(* IEC 61131-3 sources: IRIS-Project/LASAL CONTROL SOFTWARE/LasalProject_2025_09_25/Class/Automatic_Step_Settings, 1 file *)

(* ---- Automatic_Step_Settings.st ---- *)
(*!
<Class
	Name               = "Automatic_Step_Settings"
	Revision           = "0.0"
	RealtimeTask       = "false"
	CyclicTask         = "true"
	DefCyclictime      = "500 ms"
	BackgroundTask     = "false"
	Sigmatek           = "false"
	OSInterface        = "false"
	HighPriority       = "false"
	Automatic          = "false"
	UpdateMode         = "Prescan"
	SharedCommandTable = "true"
	Objectsize         = "(900,1020)">
	<Channels>
		<Server Name="ClassSvr" Visualized="false" Initialize="false" WriteProtected="true" Retentive="false"/>
		<Server Name="M1_Correction_Step" Visualized="false" Initialize="false" WriteProtected="false" Retentive="false"/>
		<Server Name="M3_Correction_Step" Visualized="false" Initialize="false" WriteProtected="false" Retentive="false"/>
		<Server Name="M4_Correction_Step" Visualized="false" Initialize="false" WriteProtected="false" Retentive="false"/>
		<Server Name="M5_ChargingCorrection_step_1" Visualized="false" Initialize="false" WriteProtected="false" Retentive="false"/>
		<Server Name="M5_ChargingCorrection_step_2" Visualized="false" Initialize="false" WriteProtected="false" Retentive="false"/>
		<Server Name="M5_ChargingCorrection_step_3" Visualized="false" Initialize="false" WriteProtected="false" Retentive="false"/>
		<Server Name="M5_DischargingCorrection_step" Visualized="false" Initialize="false" WriteProtected="false" Retentive="false"/>
		<Server Name="M5_IrradiationCorrection_step_1" Visualized="false" Initialize="false" WriteProtected="false" Retentive="false"/>
		<Server Name="M5_IrradiationCorrection_step_2" Visualized="false" Initialize="false" WriteProtected="false" Retentive="false"/>
		<Server Name="M5_IrradiationCorrection_step_3" Visualized="false" Initialize="false" WriteProtected="false" Retentive="false"/>
		<Client Name="c_M1_Correction_Step" Required="false" Internal="false"/>
		<Client Name="c_M3_Correction_Step" Required="true" Internal="false"/>
		<Client Name="c_M4_Correction_Step" Required="true" Internal="false"/>
		<Client Name="c_M5_ChargingCorrection_Step_1" Required="true" Internal="false"/>
		<Client Name="c_M5_ChargingCorrection_Step_2" Required="true" Internal="false"/>
		<Client Name="c_M5_ChargingCorrection_Step_3" Required="true" Internal="false"/>
		<Client Name="c_M5_DischargingCorrection_step" Required="true" Internal="false"/>
		<Client Name="c_M5_IrradiationCorrection_Step_1" Required="true" Internal="false"/>
		<Client Name="c_M5_IrradiationCorrection_Step_2" Required="true" Internal="false"/>
		<Client Name="c_M5_IrradiationCorrection_step_3" Required="true" Internal="false"/>
	</Channels>
	<Separators>
		<Servers>
			<SepChn Position="3"/>
			<SepChn Position="7"/>
			<SepChn Position="11"/>
			<SepChn Position="15"/>
			<SepChn Position="1"/>
			<SepChn Position="5"/>
		</Servers>
		<Clients>
			<SepChn Position="1"/>
			<SepChn Position="5"/>
			<SepChn Position="9"/>
			<SepChn Position="13"/>
			<SepChn Position="3"/>
		</Clients>
	</Separators>
</Class>
*)
Automatic_Step_Settings : CLASS
  //Servers:
	ClassSvr 	: SvrChCmd_DINT;
	M1_Correction_Step 	: SvrCh_DINT;
	M3_Correction_Step 	: SvrCh_DINT;
	M4_Correction_Step 	: SvrCh_DINT;
	M5_ChargingCorrection_step_1 	: SvrCh_DINT;
	M5_ChargingCorrection_step_2 	: SvrCh_DINT;
	M5_ChargingCorrection_step_3 	: SvrCh_DINT;
	M5_IrradiationCorrection_step_1 	: SvrCh_DINT;
	M5_IrradiationCorrection_step_2 	: SvrCh_DINT;
	M5_IrradiationCorrection_step_3 	: SvrCh_DINT;
	M5_DischargingCorrection_step 	: SvrCh_DINT;
  //Clients:
	c_M1_Correction_Step 	: CltCh_DINT;
	c_M3_Correction_Step 	: CltCh_DINT;
	c_M4_Correction_Step 	: CltCh_DINT;
	c_M5_ChargingCorrection_Step_1 	: CltCh_DINT;
	c_M5_ChargingCorrection_Step_2 	: CltCh_DINT;
	c_M5_ChargingCorrection_Step_3 	: CltCh_DINT;
	c_M5_IrradiationCorrection_Step_1 	: CltCh_DINT;
	c_M5_IrradiationCorrection_Step_2 	: CltCh_DINT;
	c_M5_IrradiationCorrection_step_3 	: CltCh_DINT;
	c_M5_DischargingCorrection_step 	: CltCh_DINT;
  //Variables:
		v_M1_CorrectionStep 	: DINT;
		v_M3_CorrectionStep 	: DINT;
		v_M5_ChargingCorrection_step_1 	: DINT;
		v_M5_ChargingCorrection_step_2 	: DINT;
		v_M5_ChargingCorrection_step_3 	: DINT;
		v_M5_IrradiationCorrection_step_1 	: DINT;
		v_M5_IrradiationCorrection_step_2 	: DINT;
		v_M5_IrradiationCorrection_step_3 	: DINT;
		v_M5_DiscahrgingCorrection_step 	: DINT;
		v_M4_CorrectionStep 	: DINT;
  //Functions:

	FUNCTION VIRTUAL GLOBAL Init;

	FUNCTION VIRTUAL GLOBAL CyWork
		VAR_INPUT
			EAX 	: UDINT;
		END_VAR
		VAR_OUTPUT
			state (EAX) 	: UDINT;
		END_VAR;

	FUNCTION VIRTUAL GLOBAL M1_Correction_Step::Read
		VAR_OUTPUT
			output (EAX) 	: DINT;
		END_VAR;

	FUNCTION VIRTUAL GLOBAL M3_Correction_Step::Read
		VAR_OUTPUT
			output (EAX) 	: DINT;
		END_VAR;

	FUNCTION VIRTUAL GLOBAL M4_Correction_Step::Read
		VAR_OUTPUT
			output (EAX) 	: DINT;
		END_VAR;

	FUNCTION VIRTUAL GLOBAL M5_ChargingCorrection_step_1::Read
		VAR_OUTPUT
			output (EAX) 	: DINT;
		END_VAR;

	FUNCTION VIRTUAL GLOBAL M5_ChargingCorrection_step_2::Read
		VAR_OUTPUT
			output (EAX) 	: DINT;
		END_VAR;

	FUNCTION VIRTUAL GLOBAL M5_ChargingCorrection_step_3::Read
		VAR_OUTPUT
			output (EAX) 	: DINT;
		END_VAR;

	FUNCTION VIRTUAL GLOBAL M5_IrradiationCorrection_step_1::Read
		VAR_OUTPUT
			output (EAX) 	: DINT;
		END_VAR;

	FUNCTION VIRTUAL GLOBAL M5_IrradiationCorrection_step_2::Read
		VAR_OUTPUT
			output (EAX) 	: DINT;
		END_VAR;

	FUNCTION VIRTUAL GLOBAL M5_IrradiationCorrection_step_3::Read
		VAR_OUTPUT
			output (EAX) 	: DINT;
		END_VAR;

	FUNCTION VIRTUAL GLOBAL M5_DischargingCorrection_step::Read
		VAR_OUTPUT
			output (EAX) 	: DINT;
		END_VAR;
  //Tables:
	FUNCTION @STD
		VAR_OUTPUT
			ret_code	: CONFSTATES;
		END_VAR;
	FUNCTION GLOBAL TAB @CT_;
END_CLASS;

FUNCTION VIRTUAL GLOBAL Automatic_Step_Settings::CyWork
	VAR_INPUT
		EAX 	: UDINT;
	END_VAR
	VAR_OUTPUT
		state (EAX) 	: UDINT;
	END_VAR

//READ FORM EPICS WITH MODBUS

  v_M1_CorrectionStep:=M1_Correction_Step.Read();

  v_M3_CorrectionStep:=M3_Correction_Step.Read();

  v_M4_CorrectionStep:=M4_Correction_Step.Read();

  v_M5_ChargingCorrection_step_1:=M5_ChargingCorrection_step_1.Read();
  v_M5_ChargingCorrection_step_2:=M5_ChargingCorrection_step_2.Read();
  v_M5_ChargingCorrection_step_3:=M5_ChargingCorrection_step_3.Read();

  v_M5_IrradiationCorrection_step_1:=M5_IrradiationCorrection_step_1.Read();
  v_M5_IrradiationCorrection_step_2:=M5_IrradiationCorrection_step_2.Read();
  v_M5_IrradiationCorrection_step_3:=M5_IrradiationCorrection_step_3.Read();

  v_M5_DiscahrgingCorrection_step:=M5_DischargingCorrection_step.Read();

//WRITE TO USE IN PLC

  c_M1_Correction_Step.Write(input:=v_M1_CorrectionStep);

  c_M3_Correction_Step.Write(input:=v_M3_CorrectionStep);

  c_M4_Correction_Step.Write(input:=v_M4_CorrectionStep);

  c_M5_ChargingCorrection_Step_1.Write(input:=v_M5_ChargingCorrection_step_1);
  c_M5_ChargingCorrection_Step_2.Write(input:=v_M5_ChargingCorrection_step_2);
  c_M5_ChargingCorrection_Step_3.Write(input:=v_M5_ChargingCorrection_step_3);

  c_M5_IrradiationCorrection_Step_1.Write(input:=v_M5_IrradiationCorrection_step_1);
  c_M5_IrradiationCorrection_Step_2.Write(input:=v_M5_IrradiationCorrection_step_2);
  c_M5_IrradiationCorrection_step_3.Write(input:=v_M5_IrradiationCorrection_step_3);

  c_M5_DischargingCorrection_step.Write(input:=v_M5_DiscahrgingCorrection_step);

	state := READY;
END_FUNCTION

FUNCTION VIRTUAL GLOBAL Automatic_Step_Settings::M5_ChargingCorrection_step_1::Read
	VAR_OUTPUT
		output (EAX) 	: DINT;
	END_VAR

	output := M5_ChargingCorrection_step_1;

END_FUNCTION

FUNCTION VIRTUAL GLOBAL Automatic_Step_Settings::M5_ChargingCorrection_step_2::Read
	VAR_OUTPUT
		output (EAX) 	: DINT;
	END_VAR

	output := M5_ChargingCorrection_step_2;

END_FUNCTION

FUNCTION VIRTUAL GLOBAL Automatic_Step_Settings::M5_ChargingCorrection_step_3::Read
	VAR_OUTPUT
		output (EAX) 	: DINT;
	END_VAR

	output := M5_ChargingCorrection_step_3;

END_FUNCTION

FUNCTION VIRTUAL GLOBAL Automatic_Step_Settings::M5_IrradiationCorrection_step_1::Read
	VAR_OUTPUT
		output (EAX) 	: DINT;
	END_VAR

	output := M5_IrradiationCorrection_step_1;

END_FUNCTION

FUNCTION VIRTUAL GLOBAL Automatic_Step_Settings::M5_IrradiationCorrection_step_2::Read
	VAR_OUTPUT
		output (EAX) 	: DINT;
	END_VAR

	output := M5_IrradiationCorrection_step_2;

END_FUNCTION

FUNCTION VIRTUAL GLOBAL Automatic_Step_Settings::M5_IrradiationCorrection_step_3::Read
	VAR_OUTPUT
		output (EAX) 	: DINT;
	END_VAR

	output := M5_IrradiationCorrection_step_3;

END_FUNCTION

FUNCTION VIRTUAL GLOBAL Automatic_Step_Settings::M5_DischargingCorrection_step::Read
	VAR_OUTPUT
		output (EAX) 	: DINT;
	END_VAR

	output := M5_DischargingCorrection_step;

END_FUNCTION

FUNCTION VIRTUAL GLOBAL Automatic_Step_Settings::M1_Correction_Step::Read
	VAR_OUTPUT
		output (EAX) 	: DINT;
	END_VAR

	output := M1_Correction_Step;

END_FUNCTION

FUNCTION VIRTUAL GLOBAL Automatic_Step_Settings::M3_Correction_Step::Read
	VAR_OUTPUT
		output (EAX) 	: DINT;
	END_VAR

	output := M3_Correction_Step;

END_FUNCTION

FUNCTION VIRTUAL GLOBAL Automatic_Step_Settings::Init

v_M1_CorrectionStep:=0;

v_M3_CorrectionStep:=0;

v_M4_CorrectionStep:=0;

v_M5_ChargingCorrection_step_1:=0;
v_M5_ChargingCorrection_step_2:=0;
v_M5_ChargingCorrection_step_3:=0;

v_M5_IrradiationCorrection_step_1:=0;
v_M5_IrradiationCorrection_step_2:=0;
v_M5_IrradiationCorrection_step_3:=0;

v_M5_DiscahrgingCorrection_step:=0;

END_FUNCTION

FUNCTION VIRTUAL GLOBAL Automatic_Step_Settings::M4_Correction_Step::Read
	VAR_OUTPUT
		output (EAX) 	: DINT;
	END_VAR

	output := M4_Correction_Step;

END_FUNCTION
